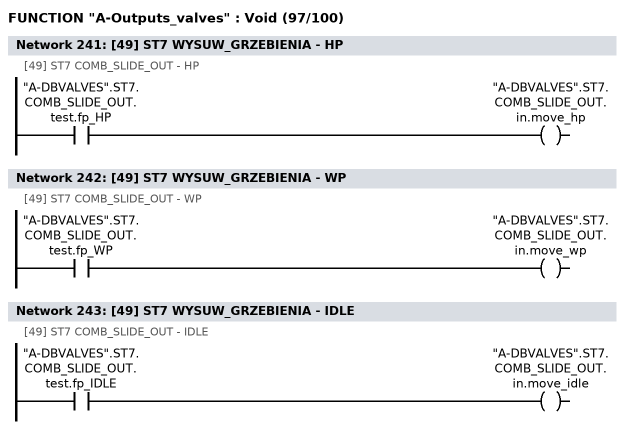
      O "A-DBVALVES".ST7.COMB_SLIDE_OUT.test.fp_HP;
//    O     "A-Flags".STATION.IN_HP_STEP
      = "A-DBVALVES".ST7.COMB_SLIDE_OUT.in.move_hp;
NETWORK
TITLE = [49] ST7 WYSUW_GRZEBIENIA - WP
//[49] ST7 COMB_SLIDE_OUT - WP
      O "A-DBVALVES".ST7.COMB_SLIDE_OUT.test.fp_WP;
      = "A-DBVALVES".ST7.COMB_SLIDE_OUT.in.move_wp;
NETWORK
TITLE = [49] ST7 WYSUW_GRZEBIENIA - IDLE
//[49] ST7 COMB_SLIDE_OUT - IDLE
      O "A-DBVALVES".ST7.COMB_SLIDE_OUT.test.fp_IDLE;
      = "A-DBVALVES".ST7.COMB_SLIDE_OUT.in.move_idle;
NETWORK
TITLE = [49] ST7 WYSUW_GRZEBIENIA
//[49] ST7 COMB_SLIDE_OUT
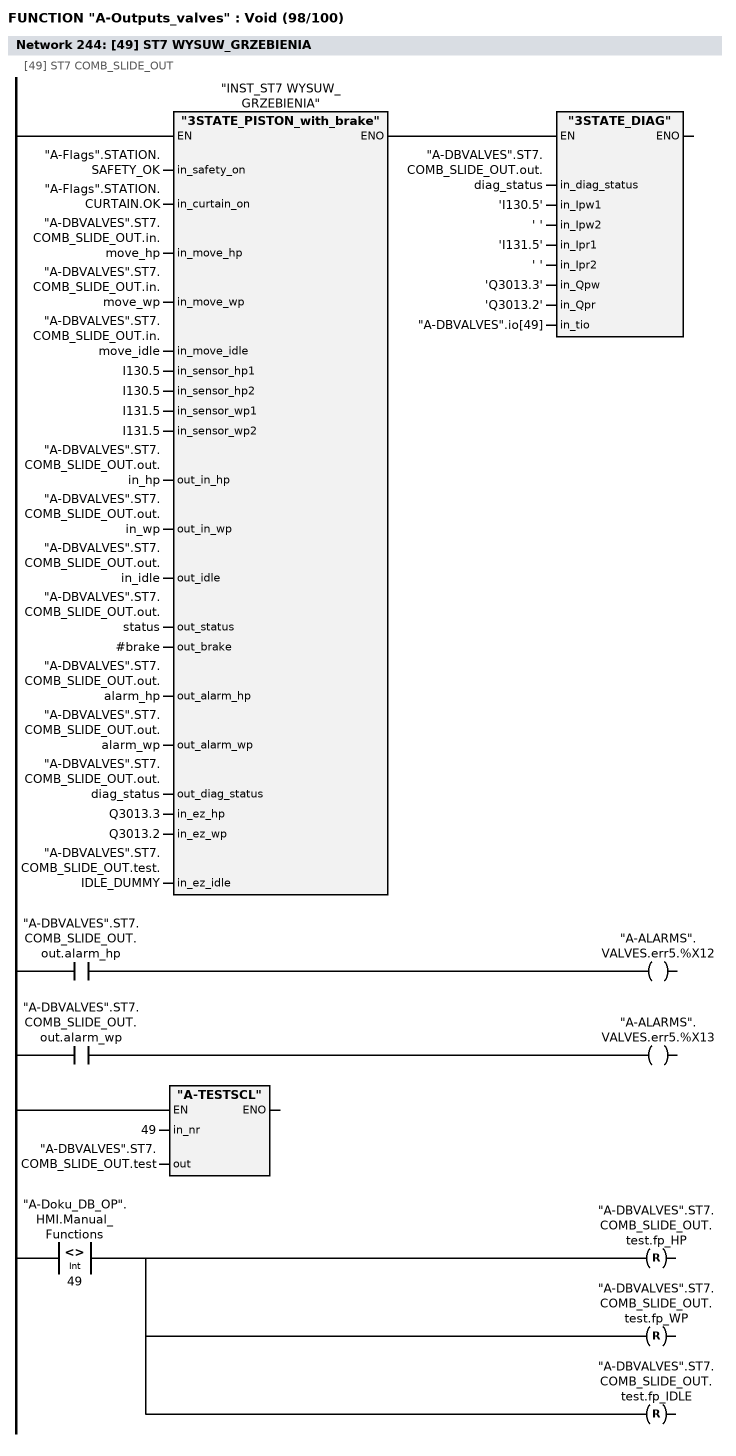
      CALL "3STATE_PISTON_with_brake", "INST_ST7 WYSUW_GRZEBIENIA"
      (  in_safety_on                := "A-Flags".STATION.SAFETY_OK ,
         in_curtain_on               := "A-Flags".STATION.CURTAIN.OK ,
         in_move_hp                  := "A-DBVALVES".ST7.COMB_SLIDE_OUT.in.move_hp ,
         in_move_wp                  := "A-DBVALVES".ST7.COMB_SLIDE_OUT.in.move_wp ,
         in_move_idle                := "A-DBVALVES".ST7.COMB_SLIDE_OUT.in.move_idle ,
         in_sensor_hp1               := I130.5 ,
         in_sensor_hp2               := I130.5 ,
         in_sensor_wp1               := I131.5 ,
         in_sensor_wp2               := I131.5 ,
         out_in_hp                   := "A-DBVALVES".ST7.COMB_SLIDE_OUT.out.in_hp ,
         out_in_wp                   := "A-DBVALVES".ST7.COMB_SLIDE_OUT.out.in_wp ,
         out_idle                    := "A-DBVALVES".ST7.COMB_SLIDE_OUT.out.in_idle ,
         out_status                  := "A-DBVALVES".ST7.COMB_SLIDE_OUT.out.status ,
         out_brake                   := #brake ,
         out_alarm_hp                := "A-DBVALVES".ST7.COMB_SLIDE_OUT.out.alarm_hp ,
         out_alarm_wp                := "A-DBVALVES".ST7.COMB_SLIDE_OUT.out.alarm_wp ,
         out_diag_status             := "A-DBVALVES".ST7.COMB_SLIDE_OUT.out.diag_status ,
         in_ez_hp                    := Q3013.3 ,
         in_ez_wp                    := Q3013.2 ,
         in_ez_idle                  := "A-DBVALVES".ST7.COMB_SLIDE_OUT.test.IDLE_DUMMY
      );

      CALL "3STATE_DIAG"
      (  in_diag_status              := "A-DBVALVES".ST7.COMB_SLIDE_OUT.out.diag_status ,
         in_Ipw1                     := 'I130.5' ,
         in_Ipw2                     := ' ' ,
         in_Ipr1                     := 'I131.5' ,
         in_Ipr2                     := ' ' ,
         in_Qpw                      := 'Q3013.3' ,
         in_Qpr                      := 'Q3013.2' ,
         in_tio                      := "A-DBVALVES".io[49]
      );

      A "A-DBVALVES".ST7.COMB_SLIDE_OUT.out.alarm_hp;
      = "A-ALARMS".VALVES.err5.%X12;

      A "A-DBVALVES".ST7.COMB_SLIDE_OUT.out.alarm_wp;
      = "A-ALARMS".VALVES.err5.%X13;

      CALL "A-TESTSCL"
      (  in_nr                       := 49 ,
         out                         := "A-DBVALVES".ST7.COMB_SLIDE_OUT.test
      );

      A(;
      L "A-Doku_DB_OP".HMI.Manual_Functions;
      L 49;
      <>I;
      );
      R "A-DBVALVES".ST7.COMB_SLIDE_OUT.test.fp_HP;
      R "A-DBVALVES".ST7.COMB_SLIDE_OUT.test.fp_WP;
      R "A-DBVALVES".ST7.COMB_SLIDE_OUT.test.fp_IDLE;
NETWORK
TITLE = -

NETWORK
TITLE = [50] ST7 GRZEBIEN - HP
//[50] ST7 COMB - HP
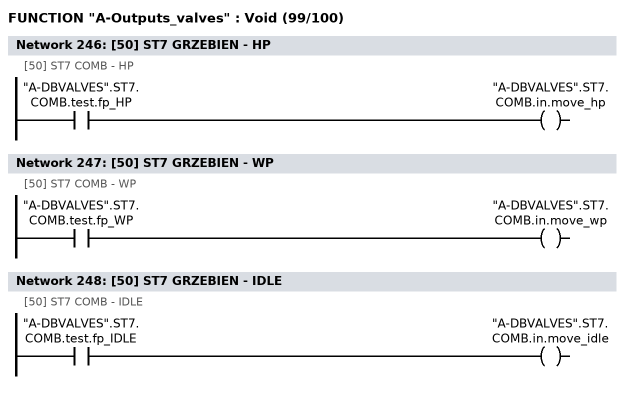
      O "A-DBVALVES".ST7.COMB.test.fp_HP;
//    O     "A-Flags".STATION.IN_HP_STEP
      = "A-DBVALVES".ST7.COMB.in.move_hp;
NETWORK
TITLE = [50] ST7 GRZEBIEN - WP
//[50] ST7 COMB - WP
      O "A-DBVALVES".ST7.COMB.test.fp_WP;
      = "A-DBVALVES".ST7.COMB.in.move_wp;
NETWORK
TITLE = [50] ST7 GRZEBIEN - IDLE
//[50] ST7 COMB - IDLE
      O "A-DBVALVES".ST7.COMB.test.fp_IDLE;
      = "A-DBVALVES".ST7.COMB.in.move_idle;
NETWORK
TITLE = [50] ST7 GRZEBIEN
//[50] ST7 COMB
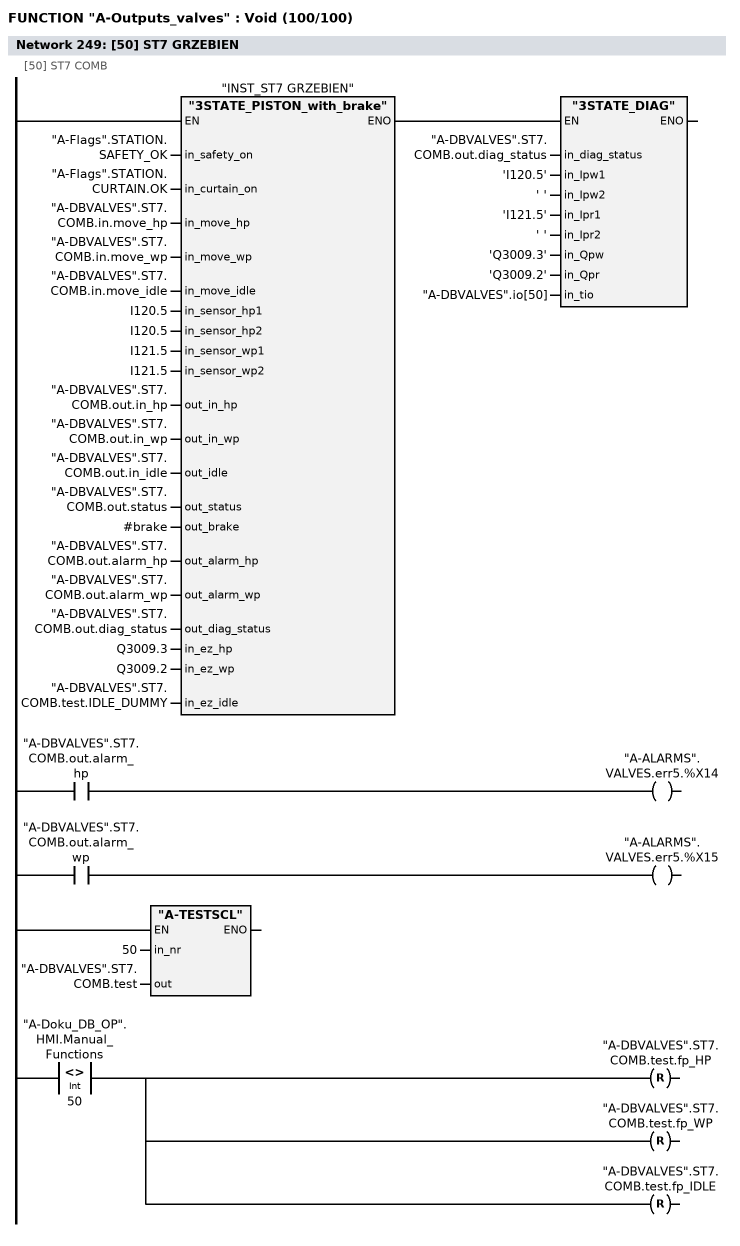
      CALL "3STATE_PISTON_with_brake", "INST_ST7 GRZEBIEN"
      (  in_safety_on                := "A-Flags".STATION.SAFETY_OK ,
         in_curtain_on               := "A-Flags".STATION.CURTAIN.OK ,
         in_move_hp                  := "A-DBVALVES".ST7.COMB.in.move_hp ,
         in_move_wp                  := "A-DBVALVES".ST7.COMB.in.move_wp ,
         in_move_idle                := "A-DBVALVES".ST7.COMB.in.move_idle ,
         in_sensor_hp1               := I120.5 ,
         in_sensor_hp2               := I120.5 ,
         in_sensor_wp1               := I121.5 ,
         in_sensor_wp2               := I121.5 ,
         out_in_hp                   := "A-DBVALVES".ST7.COMB.out.in_hp ,
         out_in_wp                   := "A-DBVALVES".ST7.COMB.out.in_wp ,
         out_idle                    := "A-DBVALVES".ST7.COMB.out.in_idle ,
         out_status                  := "A-DBVALVES".ST7.COMB.out.status ,
         out_brake                   := #brake ,
         out_alarm_hp                := "A-DBVALVES".ST7.COMB.out.alarm_hp ,
         out_alarm_wp                := "A-DBVALVES".ST7.COMB.out.alarm_wp ,
         out_diag_status             := "A-DBVALVES".ST7.COMB.out.diag_status ,
         in_ez_hp                    := Q3009.3 ,
         in_ez_wp                    := Q3009.2 ,
         in_ez_idle                  := "A-DBVALVES".ST7.COMB.test.IDLE_DUMMY
      );

      CALL "3STATE_DIAG"
      (  in_diag_status              := "A-DBVALVES".ST7.COMB.out.diag_status ,
         in_Ipw1                     := 'I120.5' ,
         in_Ipw2                     := ' ' ,
         in_Ipr1                     := 'I121.5' ,
         in_Ipr2                     := ' ' ,
         in_Qpw                      := 'Q3009.3' ,
         in_Qpr                      := 'Q3009.2' ,
         in_tio                      := "A-DBVALVES".io[50]
      );

      A "A-DBVALVES".ST7.COMB.out.alarm_hp;
      = "A-ALARMS".VALVES.err5.%X14;

      A "A-DBVALVES".ST7.COMB.out.alarm_wp;
      = "A-ALARMS".VALVES.err5.%X15;

      CALL "A-TESTSCL"
      (  in_nr                       := 50 ,
         out                         := "A-DBVALVES".ST7.COMB.test
      );

      A(;
      L "A-Doku_DB_OP".HMI.Manual_Functions;
      L 50;
      <>I;
      );
      R "A-DBVALVES".ST7.COMB.test.fp_HP;
      R "A-DBVALVES".ST7.COMB.test.fp_WP;
      R "A-DBVALVES".ST7.COMB.test.fp_IDLE;
NETWORK
TITLE = -


END_FUNCTION

